{attribute 'conditionalshow'}
FUNCTION_BLOCK FB_CV_SINT_TO_WORD
VAR_INPUT
	{attribute 'hide'}
	siInputValue_1				: SINT;								//Input value that is converted into the output value	
	{attribute 'hide'}						
	siInputValue_2				: SINT;								//Input value that is converted into the output value
	{attribute 'hide'}
	eByteOrderForConvert		: eByteOrder;						//Byte Format
END_VAR
VAR_OUTPUT
	{attribute 'hide'}
	wOutputValue				: WORD;								//Converted output value
END_VAR
VAR
END_VAR

//Creator : Kai Ebensperger
//Company : Lynus AG
//Date : 28.04.2021
//Version : 1.0.0.0

//With this functionblock its possible to convert a certain Datatyp in a other Datatype
//The byte order can be selected between BigEndian and LittleEndian
//SINT TO WORD
//Created for the Edge Device Lib over Modbus TCP
//Modbus TCP is WORD oriented

IF eByteOrderForConvert = eByteOrder.eBigEndian THEN
	wOutputValue := SHL(BYTE_TO_WORD(SINT_TO_BYTE(siInputValue_1)),8) + BYTE_TO_WORD(SINT_TO_BYTE(siInputValue_2));
ELSE
	wOutputValue := SHL(BYTE_TO_WORD(SINT_TO_BYTE(siInputValue_2)),8) + BYTE_TO_WORD(SINT_TO_BYTE(siInputValue_1));
END_IF

END_FUNCTION_BLOCK

(* stored: Version 1.1.0.1, ProductVersion 3.1.4024.9
   POU FB_CV_SINT_TO_WORD: Id {4b1eeb78-5a84-4b8e-9f8f-dac2ccd99114}, SpecialFunc None *)
